{attribute 'enable_dynamic_creation'}
FUNCTION_BLOCK OpcUaMethodCallRequestItem EXTENDS OpcUaRequestItem
VAR_STAT
	//! <summary>Class name shared by all instances of this function block.</summary>
	_ClassName : STRING := __POUNAME();
END_VAR
VAR
	_ObjectNamespaceUri : STRING(Tc2_System.MAX_STRING_LENGTH);
	_ObjectNodeId: Tc3_PLCopen_OpcUa.ST_UANodeID;		
	_ObjectNamespaceIndexValid : BOOL;

	_MethodNamespaceUri : STRING(Tc2_System.MAX_STRING_LENGTH);
	_MethodNodeId: Tc3_PLCopen_OpcUa.ST_UANodeID;		
	_MethodNamespaceIndexValid : BOOL;

	_NumberOfReceivedBytesCount : POINTER TO UDINT;
	
	_GetMethodHandle : Tc3_PLCopen_OpcUa.UA_MethodGetHandle;
	_MethodCall : Tc3_PLCopen_OpcUa.UA_MethodCall;
	_ReleaseMethodHandle : Tc3_PLCopen_OpcUa.UA_MethodReleaseHandle;	
END_VAR

{attribute 'monitoring' := 'call'}
PROPERTY ClassName : REFERENCE TO STRING
GET
ClassName REF= _ClassName;
END_GET
END_PROPERTY

METHOD GetHandle : OPC_UA_ACTION_EXECUTION_STATE
VAR_INPUT
	connectionHandle : DWORD;
END_VAR
VAR_OUTPUT
	exception : Exception;
END_VAR
_ConnectionHandle := connectionHandle;

GetHandle := OPC_UA_ACTION_EXECUTION_STATE.DONE;
	
IF NOT _ObjectNamespaceIndexValid THEN
	ExceptionHelper.Throw(
		0,
		WString.Concat3(
			"UA__GetMethodHandle error: invalid object namespace index for namespace '",
			TO_WSTRING(_ObjectNamespaceUri),
			"'"
		),
		__POUNAME(),
		ClassName,
		CurrentNamespace.Name,
		__POSITION(
	)
	);
	GetHandle := OPC_UA_ACTION_EXECUTION_STATE.ERROR;				
	AdsLogger.LogMessage(
		LOGGING_LEVEL.INFORMATION,
		WString.Concat3(
			"---OpcUaRequest GetNodeHandle error: invalid object namespace index for namespace '",
			TO_WSTRING(_ObjectNamespaceUri),
			"'"
		)
	);
ELSIF NOT _MethodNamespaceIndexValid THEN
	ExceptionHelper.Throw(
		0,
		WString.Concat3(
			"UA__GetMethodHandle error: invalid method namespace index for namespace '",
			TO_WSTRING(_MethodNamespaceUri),
			"'"
		),
		__POUNAME(),
		ClassName,
		CurrentNamespace.Name,
		__POSITION(
	)
	);
	GetHandle := OPC_UA_ACTION_EXECUTION_STATE.ERROR;				
	AdsLogger.LogMessage(
		LOGGING_LEVEL.INFORMATION,
		WString.Concat3(
			"---OpcUaRequest GetMethodHandle error: invalid method namespace index for namespace '",
			TO_WSTRING(_MethodNamespaceUri),
			"'"
		)
	);
ELSE
	_GetMethodHandle(Execute := TRUE, ConnectionHdl := _ConnectionHandle, ObjectNodeID := _ObjectNodeId, MethodNodeID := _MethodNodeId);

	IF _GetMethodHandle.Error THEN
		ExceptionHelper.Throw(
		_GetMethodHandle.ErrorID,
		WString.Concat7(
				"UA_GetMethodHandle error ",
				TO_WSTRING(_GetMethodHandle.ErrorID),
				" (ObjectNodeID='",
				TO_WSTRING(_ObjectNodeId.sIdentifier),
				"', MethodNodeID='",
				TO_WSTRING(_MethodNodeId.sIdentifier),
				"')"
			),
		__POUNAME(),
		ClassName,
		CurrentNamespace.Name,
		__POSITION(
	)
		);
		GetHandle := OPC_UA_ACTION_EXECUTION_STATE.ERROR;					
		AdsLogger.LogMessage(
			LOGGING_LEVEL.INFORMATION,
			WString.Concat3(
				"---OpcUaRequest GetMethodHandle error: ",
				"UA_GetMethodHandle error ",
				TO_WSTRING(_GetMethodHandle.ErrorID)
			)
		);
	ELSIF _GetMethodHandle.Busy THEN
		GetHandle := OPC_UA_ACTION_EXECUTION_STATE.BUSY;			
	END_IF
END_IF
END_METHOD

//!<param name="objectNamespaceUri">empty string if index used</param>

//!<param name="objectNamespaceIndex">zero if namespace uri used</param>

//!<param name="methodNamespaceUri">empty string if index used</param>

//!<param name="methodNamespaceIndex">zero if namespace uri used</param>

METHOD Initialize
VAR_INPUT
	objectNamespaceUri : STRING(Tc2_System.MAX_STRING_LENGTH); 
	objectNamespaceIndex : UINT; 
	objectIdentifierType : Tc3_PLCopen_OpcUa.E_UAIdentifierType;
	objectIdentifier : STRING(Tc2_System.MAX_STRING_LENGTH);	
	methodNamespaceUri : STRING(Tc2_System.MAX_STRING_LENGTH); 
	methodNamespaceIndex : UINT; 
	methodIdentifierType : Tc3_PLCopen_OpcUa.E_UAIdentifierType;
	methodIdentifier : STRING(Tc2_System.MAX_STRING_LENGTH);
	inputArgumentInfosAddress : POINTER TO ST_UAMethodArgInfo;
	inputArgumentInfosSize : UDINT;
	inputConstantArgumentsAddress : PVOID;
	inputConstantArgumentsSize : UDINT;
	inputDynamicArgumentsAddress : PVOID;
	inputDynamicArgumentsSize : UDINT;
	outputArgumentInfosAddress : POINTER TO ST_UAMethodArgInfo;
	outputArgumentInfosSize : UDINT;
	outputArgumentsInfoAndDataAddress : POINTER TO OPC_UA_OUTPUT_ARGUMENT_INFO_AND_DATA;
	outputArgumentsInfoAndDataSize : UDINT;
	numberOfReceivedBytesCount : POINTER TO UDINT;
	operationTimeout : TIME := Tc2_System.DEFAULT_ADS_TIMEOUT;
END_VAR
IF objectNamespaceUri <> '' THEN
	_ObjectNamespaceUri := objectNamespaceUri;
	_ObjectNodeId.nNamespaceIndex := 0;
	_ObjectNamespaceIndexValid := FALSE;
ELSE
	_ObjectNamespaceUri := '';
	_ObjectNodeId.nNamespaceIndex := objectNamespaceIndex;
	_ObjectNamespaceIndexValid := TRUE;
END_IF

_ObjectNodeId.eIdentifierType := objectIdentifierType;
_ObjectNodeId.sIdentifier := objectIdentifier;

IF methodNamespaceUri <> '' THEN
	_MethodNamespaceUri := methodNamespaceUri;
	_MethodNodeId.nNamespaceIndex := 0;
	_MethodNamespaceIndexValid := FALSE;
ELSE
	_MethodNamespaceUri := '';
	_MethodNodeId.nNamespaceIndex := methodNamespaceIndex;
	_MethodNamespaceIndexValid := TRUE;
END_IF

_MethodNodeId.eIdentifierType := methodIdentifierType;
_MethodNodeId.sIdentifier := methodIdentifier;
_MethodCall.nNumberOfInputArguments := inputArgumentInfosSize / SIZEOF(ST_UAMethodArgInfo);
_MethodCall.pInputArgInfo := inputArgumentInfosAddress;
_MethodCall.cbInputArgInfo := inputArgumentInfosSize;
_MethodCall.pInputArgData := inputConstantArgumentsAddress;
_MethodCall.cbInputArgData := inputConstantArgumentsSize;
_MethodCall.pInputWriteData := inputDynamicArgumentsAddress;
_MethodCall.cbInputWriteData := inputDynamicArgumentsSize;
_MethodCall.nNumberOfOutputArguments := outputArgumentInfosSize / SIZEOF(ST_UAMethodArgInfo);
_MethodCall.pOutputArgInfo := outputArgumentInfosAddress;
_MethodCall.cbOutputArgInfo := outputArgumentInfosSize;
_MethodCall.pOutputArgInfoAndData := outputArgumentsInfoAndDataAddress;
_MethodCall.cbOutputArgInfoAndData := outputArgumentsInfoAndDataSize;

_NumberOfReceivedBytesCount := numberOfReceivedBytesCount;

_GetMethodHandle.Timeout := operationTimeout;
_MethodCall.Timeout := operationTimeout;
_ReleaseMethodHandle.Timeout := operationTimeout;
END_METHOD

METHOD PerformAction : OPC_UA_ACTION_EXECUTION_STATE
VAR_OUTPUT
	exception : Exception;
END_VAR
PerformAction := OPC_UA_ACTION_EXECUTION_STATE.DONE;

_MethodCall(Execute := TRUE, ConnectionHdl := _ConnectionHandle, MethodHdl := _GetMethodHandle.MethodHdl);
		
IF _MethodCall.Error THEN
	ExceptionHelper.Throw(
		_GetMethodHandle.ErrorID,
		WString.Concat7(
			"UA_MethodCall error ",
			TO_WSTRING(_MethodCall.ErrorID),
			" (ObjectNodeID='",
			TO_WSTRING(_ObjectNodeId.sIdentifier),
			"', MethodNodeID='",
			TO_WSTRING(_MethodNodeId.sIdentifier),
			"')"
		),
		__POUNAME(),
		ClassName,
		CurrentNamespace.Name,
		__POSITION(
	)
	);
	PerformAction := OPC_UA_ACTION_EXECUTION_STATE.ERROR;			
	AdsLogger.LogMessage(
		LOGGING_LEVEL.INFORMATION,
		WString.Concat3(
			"---OpcUaRequest PerformAction error: ",
			"UA_MethodCall error ",
			TO_WSTRING(_MethodCall.ErrorID)
		)
	);
ELSIF _MethodCall.Busy THEN
	PerformAction := OPC_UA_ACTION_EXECUTION_STATE.BUSY;
ELSIF _GetMethodHandle.Done AND_THEN _NumberOfReceivedBytesCount <> 0 THEN
 	_NumberOfReceivedBytesCount^ := _MethodCall.cbRead_R;
END_IF
END_METHOD

METHOD ReleaseHandle : OPC_UA_ACTION_EXECUTION_STATE
VAR_OUTPUT
	exception : Exception;
END_VAR
ReleaseHandle := OPC_UA_ACTION_EXECUTION_STATE.DONE;
	
_ReleaseMethodHandle(Execute := TRUE, ConnectionHdl := _ConnectionHandle, MethodHdl := _GetMethodHandle.MethodHdl);

IF _ReleaseMethodHandle.Error THEN
	ExceptionHelper.Throw(
		_ReleaseMethodHandle.ErrorID,
		WCONCAT("UA_ReleaseMethodHandle error ", TO_WSTRING(_ReleaseMethodHandle.ErrorID)),
		__POUNAME(),
		ClassName,
		CurrentNamespace.Name,
		__POSITION(
	)
	);
	ReleaseHandle := OPC_UA_ACTION_EXECUTION_STATE.ERROR;			
	AdsLogger.LogMessage(
		LOGGING_LEVEL.INFORMATION,
		WString.Concat3(
			"---OpcUaRequest ReleaseMethodHandle error: ",
			"UA_ReleaseMethodHandle error ",
			TO_WSTRING(_ReleaseMethodHandle.ErrorID)
		)
	);
ELSIF _ReleaseMethodHandle.Busy THEN
	ReleaseHandle := OPC_UA_ACTION_EXECUTION_STATE.BUSY;			
END_IF
END_METHOD

METHOD Reset
_GetMethodHandle(Execute := FALSE);
ResetAction();
_ReleaseMethodHandle(Execute := FALSE);
END_METHOD

METHOD ResetAction
_MethodCall(Execute := FALSE);
END_METHOD

METHOD SetNamespaceIndexForNamespaceUri
VAR_INPUT
	namespaceUri : STRING(Tc2_System.MAX_STRING_LENGTH);
	namespaceIndex : UINT;
END_VAR
IF NOT _ObjectNamespaceIndexValid AND_THEN _ObjectNamespaceUri = namespaceUri THEN
	_ObjectNodeId.nNamespaceIndex := namespaceIndex;
	_ObjectNamespaceIndexValid := TRUE;					
END_IF

IF NOT _MethodNamespaceIndexValid AND_THEN _MethodNamespaceUri = namespaceUri THEN
	_MethodNodeId.nNamespaceIndex := namespaceIndex;
	_MethodNamespaceIndexValid := TRUE;					
END_IF
END_METHOD

END_FUNCTION_BLOCK

(* stored: Version 1.1.0.1
   POU OpcUaMethodCallRequestItem: Id {1ce9736d-a860-43ea-b628-99cef6edb8d1}, SpecialFunc None
   Property ClassName: Id {0367600d-2c3d-4938-b800-22a3e07d4ddc}
   Get Get: Id {2e212076-844e-48a3-a008-0569d42bd65a}
   Method GetHandle: Id {dcea29b7-b286-4c8e-9bda-1ac4ca8b53fa}
   Method Initialize: Id {8c789994-1dce-4457-a3d0-e13a3ea4b2b6}
   Method PerformAction: Id {c63aaae3-f356-41fa-b31c-fc78704b0a15}
   Method ReleaseHandle: Id {8bc2bf16-99bf-488f-8bbf-846088c501ac}
   Method Reset: Id {1da02c69-4ec4-4da2-94d5-c953bf4b9a76}
   Method ResetAction: Id {9e553769-2b03-4812-9c99-a1b35979b0ed}
   Method SetNamespaceIndexForNamespaceUri: Id {b904cfec-751c-4a67-94ed-ab556a660a02} *)
